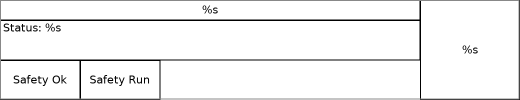
VISUALIZATION UI_StandardRoom  // 520x100
VAR_IN_OUT
	pou			: TempRoom;
END_VAR
    Rectangle (0,0 420x20), "%s", text variable: CONCAT('Room', pou._room._nId )
    Rectangle (0,20 420x40), "Status: %s", text variable: pou._ctx.hmi.sStatusText
        p55702900: pou._ctx.hmi.nStatusColor
    Rectangle (420,0 100x100), "%s", text variable: pou._ctx.hmi.sButtonText, invisible if: pou._hmi.bHideReset
        toggle pou._hmi.bReset
    Rectangle (0,60 80x40), "Safety Ok", colour toggle: pou.bSafetyOk
        toggle pou.bSafetyOk
    Rectangle (80,60 80x40), "Safety Run", colour toggle: pou.bSafetyRun
        toggle pou.bSafetyRun
END_VISUALIZATION

(* stored: Version 1.1.0.1
   Visu UI_StandardRoom: Id {c568871d-7da9-43be-9c34-308759e688ca} *)
